FUNCTION_BLOCK PiscaPisca
VAR_INPUT
	Iniciar: BOOL;
	SinalOn: TIME := T#1s;
	SinalOff: TIME := T#1s;
END_VAR
VAR_OUTPUT
	Saida: BOOL;
END_VAR
VAR
	T1: TON;
	T2: TON;
END_VAR

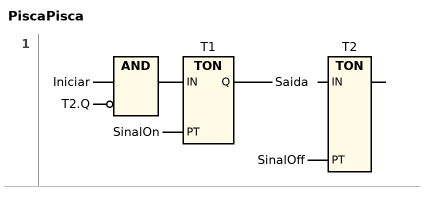
// NETWORK 1
T1(IN := Iniciar AND NOT T2.Q, PT := SinalOn); // TON
Saida := T1.Q;
T2(IN := T1.Q, PT := SinalOff); // TON

END_FUNCTION_BLOCK

(* stored: Version 1.1.0.1
   POU PiscaPisca: Id {15de89fd-9f37-4ad3-bc23-74d883f3698e}, SpecialFunc None *)
